_CFC_ (* Continuous Function Chart, elements in execution order *)
#0 OR(SCHU_P2_2_YA3_UP_RESET, SCHU_P2_2_SB)
#1 SEL(SCHU_P2_2_YA3_AI2_FILTER_ON, T#0ms, T#2s)
#2 fb_YA3:ISTOK_ANALOGVH(enable: TRUE, rawValue: SCHU_P2_2_YA3_AI2, reset: #0, enableLimitCtrl: TRUE, ctrlVoltage: NOT SCHU_P2_2_YA3_AI2_CVOLT, changeValueWithoutPower: TRUE, highRange: YA_HIGHRANGE, lowRange: YA_LOWRANGE, highLimit: SCHU_P2_2_YA_HIGHLIMIT, lowLimit: SCHU_P2_2_YA_LOWLIMIT, filterTime: #1, offset: ofset, delayEnable: YA_DELAY)
#3 SCHU_P2_2_YA3_UP_VN <= #2.presentValue
#4 SCHU_P2_2_YA3_UP_DOST <= #2.reliability
#5 Lt_otkr_zakr:ISTOK_LT(dost: #2.reliability, x: #2.presentValue, ust: 5, shkal: -, gist: 3)
#6 SCHU_P2_2_YA3_ZKR <= #5.Xm
#7 gt_otkr_otr:ISTOK_GT(dost: #2.reliability, x: #2.presentValue, ust: 95, shkal: -, gist: 3)
#8 SCHU_P2_2_YA3_OTK <= #7.Xb
#9 SUB(YA3_UST_VKL_STER_REG, YA3_UST_OTKL_STER_REG)
#10 fb_YA3bUST_VKL_STER_REG:ISTOK_GT(dost: #2.reliability, x: #2.presentValue, ust: YA3_UST_VKL_STER_REG, shkal: -, gist: #9)
#11 SCHU_P2_2_YA3_B_UST_VKL_STER_REG <= #10.Xb
#12 SCHU_P2_2_YA3_M_UST_VKL_STER_REG <= #10.XbN
#13 SUB(YA3_UST_OTKL_UVEL_CHAST, YA3_UST_VKL_UVEL_CHAST)
#14 fb_YA3mOTKL_STER_REG:ISTOK_LT(dost: #2.reliability, x: #2.presentValue, ust: YA3_UST_VKL_UVEL_CHAST, shkal: -, gist: #13)
#15 SCHU_P2_2_YA3_M_UST_VKL_UVEL_CHAST <= #14.Xm
#16 SCHU_P2_2_YA3_B_UST_VKL_UVEL_CHAST <= #14.XmN
_END_CFC_
(* the same logic as Structured Text *)
fb_YA3(enable := TRUE, rawValue := SCHU_P2_2_YA3_AI2, reset := SCHU_P2_2_YA3_UP_RESET OR SCHU_P2_2_SB, enableLimitCtrl := TRUE, ctrlVoltage := NOT SCHU_P2_2_YA3_AI2_CVOLT, changeValueWithoutPower := TRUE, highRange := YA_HIGHRANGE, lowRange := YA_LOWRANGE, highLimit := SCHU_P2_2_YA_HIGHLIMIT, lowLimit := SCHU_P2_2_YA_LOWLIMIT, filterTime := SEL(SCHU_P2_2_YA3_AI2_FILTER_ON, T#0ms, T#2s), offset := ofset, delayEnable := YA_DELAY);
SCHU_P2_2_YA3_UP_VN := fb_YA3.presentValue;
SCHU_P2_2_YA3_UP_DOST := fb_YA3.reliability;
Lt_otkr_zakr(dost := fb_YA3.reliability, x := fb_YA3.presentValue, ust := 5, gist := 3);
SCHU_P2_2_YA3_ZKR := Lt_otkr_zakr.Xm;
gt_otkr_otr(dost := fb_YA3.reliability, x := fb_YA3.presentValue, ust := 95, gist := 3);
SCHU_P2_2_YA3_OTK := gt_otkr_otr.Xb;
fb_YA3bUST_VKL_STER_REG(dost := fb_YA3.reliability, x := fb_YA3.presentValue, ust := YA3_UST_VKL_STER_REG, gist := YA3_UST_VKL_STER_REG - YA3_UST_OTKL_STER_REG);
SCHU_P2_2_YA3_B_UST_VKL_STER_REG := fb_YA3bUST_VKL_STER_REG.Xb;
SCHU_P2_2_YA3_M_UST_VKL_STER_REG := fb_YA3bUST_VKL_STER_REG.XbN;
fb_YA3mOTKL_STER_REG(dost := fb_YA3.reliability, x := fb_YA3.presentValue, ust := YA3_UST_VKL_UVEL_CHAST, gist := YA3_UST_OTKL_UVEL_CHAST - YA3_UST_VKL_UVEL_CHAST);
SCHU_P2_2_YA3_M_UST_VKL_UVEL_CHAST := fb_YA3mOTKL_STER_REG.Xm;
SCHU_P2_2_YA3_B_UST_VKL_UVEL_CHAST := fb_YA3mOTKL_STER_REG.XmN;
END_PROGRAM

(* POU Input/AI/YA4_POS, CFC *)
PROGRAM YA4_POS
VAR
	fb_YA4: ISTOK_ANALOGVH;
	ofset: REAL;
	Lt_otkr_zakr: ISTOK_LT;
	gt_otkr_otr: ISTOK_GT;
	fb_YA4mOTKL_STER_REG: ISTOK_LT;
	fb_YA4bUST_VKL_STER_REG: ISTOK_GT;
END_VAR
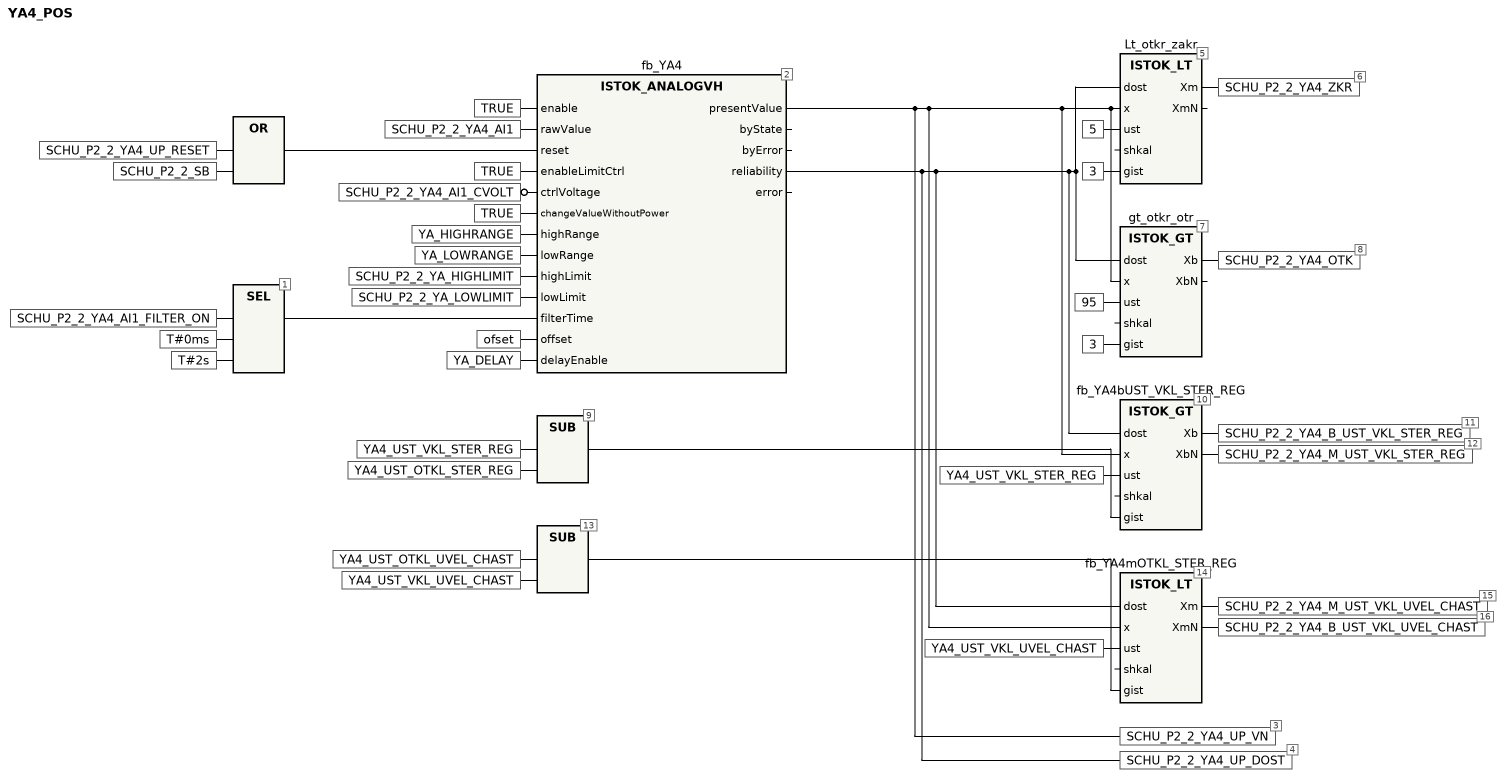
_CFC_ (* Continuous Function Chart, elements in execution order *)
#0 OR(SCHU_P2_2_YA4_UP_RESET, SCHU_P2_2_SB)
#1 SEL(SCHU_P2_2_YA4_AI1_FILTER_ON, T#0ms, T#2s)
#2 fb_YA4:ISTOK_ANALOGVH(enable: TRUE, rawValue: SCHU_P2_2_YA4_AI1, reset: #0, enableLimitCtrl: TRUE, ctrlVoltage: NOT SCHU_P2_2_YA4_AI1_CVOLT, changeValueWithoutPower: TRUE, highRange: YA_HIGHRANGE, lowRange: YA_LOWRANGE, highLimit: SCHU_P2_2_YA_HIGHLIMIT, lowLimit: SCHU_P2_2_YA_LOWLIMIT, filterTime: #1, offset: ofset, delayEnable: YA_DELAY)
#3 SCHU_P2_2_YA4_UP_VN <= #2.presentValue
#4 SCHU_P2_2_YA4_UP_DOST <= #2.reliability
#5 Lt_otkr_zakr:ISTOK_LT(dost: #2.reliability, x: #2.presentValue, ust: 5, shkal: -, gist: 3)
#6 SCHU_P2_2_YA4_ZKR <= #5.Xm
#7 gt_otkr_otr:ISTOK_GT(dost: #2.reliability, x: #2.presentValue, ust: 95, shkal: -, gist: 3)
#8 SCHU_P2_2_YA4_OTK <= #7.Xb
#9 SUB(YA4_UST_VKL_STER_REG, YA4_UST_OTKL_STER_REG)
#10 fb_YA4bUST_VKL_STER_REG:ISTOK_GT(dost: #2.reliability, x: #2.presentValue, ust: YA4_UST_VKL_STER_REG, shkal: -, gist: #9)
#11 SCHU_P2_2_YA4_B_UST_VKL_STER_REG <= #10.Xb
#12 SCHU_P2_2_YA4_M_UST_VKL_STER_REG <= #10.XbN
#13 SUB(YA4_UST_OTKL_UVEL_CHAST, YA4_UST_VKL_UVEL_CHAST)
#14 fb_YA4mOTKL_STER_REG:ISTOK_LT(dost: #2.reliability, x: #2.presentValue, ust: YA4_UST_VKL_UVEL_CHAST, shkal: -, gist: #13)
#15 SCHU_P2_2_YA4_M_UST_VKL_UVEL_CHAST <= #14.Xm
#16 SCHU_P2_2_YA4_B_UST_VKL_UVEL_CHAST <= #14.XmN
_END_CFC_
(* the same logic as Structured Text *)
fb_YA4(enable := TRUE, rawValue := SCHU_P2_2_YA4_AI1, reset := SCHU_P2_2_YA4_UP_RESET OR SCHU_P2_2_SB, enableLimitCtrl := TRUE, ctrlVoltage := NOT SCHU_P2_2_YA4_AI1_CVOLT, changeValueWithoutPower := TRUE, highRange := YA_HIGHRANGE, lowRange := YA_LOWRANGE, highLimit := SCHU_P2_2_YA_HIGHLIMIT, lowLimit := SCHU_P2_2_YA_LOWLIMIT, filterTime := SEL(SCHU_P2_2_YA4_AI1_FILTER_ON, T#0ms, T#2s), offset := ofset, delayEnable := YA_DELAY);
SCHU_P2_2_YA4_UP_VN := fb_YA4.presentValue;
SCHU_P2_2_YA4_UP_DOST := fb_YA4.reliability;
Lt_otkr_zakr(dost := fb_YA4.reliability, x := fb_YA4.presentValue, ust := 5, gist := 3);
SCHU_P2_2_YA4_ZKR := Lt_otkr_zakr.Xm;
gt_otkr_otr(dost := fb_YA4.reliability, x := fb_YA4.presentValue, ust := 95, gist := 3);
SCHU_P2_2_YA4_OTK := gt_otkr_otr.Xb;
fb_YA4bUST_VKL_STER_REG(dost := fb_YA4.reliability, x := fb_YA4.presentValue, ust := YA4_UST_VKL_STER_REG, gist := YA4_UST_VKL_STER_REG - YA4_UST_OTKL_STER_REG);
SCHU_P2_2_YA4_B_UST_VKL_STER_REG := fb_YA4bUST_VKL_STER_REG.Xb;
SCHU_P2_2_YA4_M_UST_VKL_STER_REG := fb_YA4bUST_VKL_STER_REG.XbN;
fb_YA4mOTKL_STER_REG(dost := fb_YA4.reliability, x := fb_YA4.presentValue, ust := YA4_UST_VKL_UVEL_CHAST, gist := YA4_UST_OTKL_UVEL_CHAST - YA4_UST_VKL_UVEL_CHAST);
SCHU_P2_2_YA4_M_UST_VKL_UVEL_CHAST := fb_YA4mOTKL_STER_REG.Xm;
SCHU_P2_2_YA4_B_UST_VKL_UVEL_CHAST := fb_YA4mOTKL_STER_REG.XmN;
END_PROGRAM

(* POU Input/CI/M1_OB, CFC *)
PROGRAM M1_OB
VAR
	fb_M1_OBRbSM: ISTOK_GT;
	fb_M1b30: ISTOK_GT;
	fb_M1_OBRb45: ISTOK_GT;
	fb_M1_OBRm0_1: ISTOK_LT;
	fb_M_OBR: ISTOK_ANALOGVH;
	ofset: INT := 0;
	SR_DOST_M1: RS;
	dost_ton: TON;
END_VAR
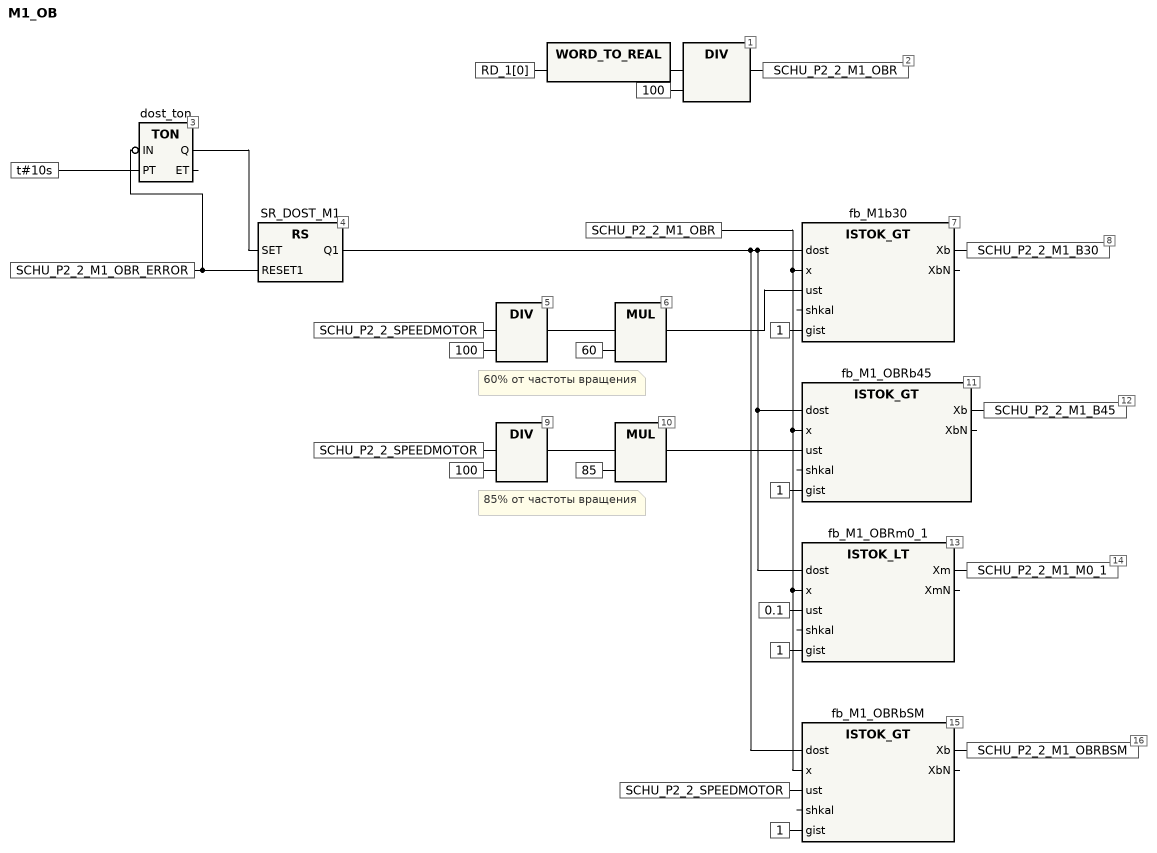
